(* PLC project Generated.project, CODESYS CODESYS V3.5 SP19 Patch 1 *)
(* stored: creationDateTime 2026-09-06T13:00:42.495836, modificationDateTime 2026-09-06T13:00:42.495836 *)

(* values of E_TranslationTraceBlockReason: NONE: ✅ Aucun blocage — permis de mouvement effectif; POWER_CUTOFF: 🧨 Coupure puissance amont (instSafetyTranslationM3.PowerCutOff) — priorité max; SAFESTOP: 🟧 SafeStop effectif (InputModule OR safety M3); SAFETY_FAULT: 🛡️ Défaut safety M3 latched (FB_Safety_Translation.Fault.Error); HEIGHT_INTERLOCK: 🚧 Interlock hauteur M1/M2 actif (risque collision); DRIVE_UNAVAILABLE: 📡 Variateur AC600 injoignable / non opérationnel; FINAL_INTERLOCK: 🛑 Barrière finale en défaut (frein / redémarrage); FAULT: ❌ Défaut mouvement M3 latched (FB_Translation.Fault.Error) *)

{attribute 'qualified_only'}
{attribute 'strict'}
TYPE E_TranslationTraceBlockReason : (NONE := 0, POWER_CUTOFF := 1, SAFESTOP := 2, SAFETY_FAULT := 3, HEIGHT_INTERLOCK := 4, DRIVE_UNAVAILABLE := 5, FINAL_INTERLOCK := 6, FAULT := 7);
END_TYPE
